// SIMATIC S7-200 project (STEP 7-Micro/WIN), CPU 221 REL 01.10

SYMBOL_TABLE USER1
start            I0.0     // start
Estop            I0.4     // stop
s1               I0.1     // cam bien hop
s2               I0.2     // cam bien dem tao
BTH              Q0.0     // bang tai hop
BTT              Q0.1     // bang tai tao
s3               I0.3     // cam bien tao
END_SYMBOL_TABLE

ORGANIZATION_BLOCK MAIN:OB1
TITLE=PROGRAM COMMENTS
BEGIN
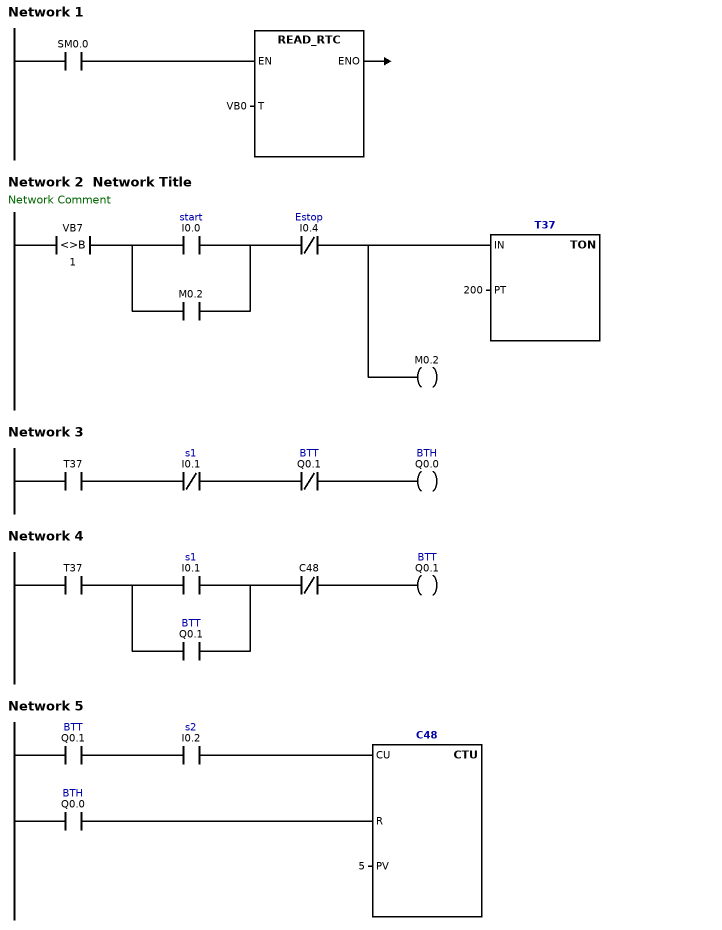
Network 1
LD     SM0.0
TODR   VB0
Network 2 // Network Title
// Network Comment
LDB<>  VB7, 1
LD     start:I0.0
O      M0.2
ALD
AN     Estop:I0.4
TON    T37, 200
=      M0.2
Network 3
LD     T37
AN     s1:I0.1
AN     BTT:Q0.1
=      BTH:Q0.0
Network 4
LD     T37
LD     s1:I0.1
O      BTT:Q0.1
ALD
AN     C48
=      BTT:Q0.1
Network 5
LD     BTT:Q0.1
A      s2:I0.2
LD     BTH:Q0.0
CTU    C48, 5
END_ORGANIZATION_BLOCK
